// TIA Portal V20 export
TYPE "LKinCtrl_typeCartesianPosition"
   STRUCT
      x : LReal;   // X
      y : LReal;   // Y
      z : LReal;   // Z
      "a" : LReal;   // A
      "b" : LReal;   // B
      c : LReal;   // C
   END_STRUCT;
END_TYPE
